FUNCTION_BLOCK INTERNAL FB_State3 EXTENDS FB_State
VAR_INPUT
END_VAR
VAR_OUTPUT
END_VAR
VAR
END_VAR

END_FUNCTION_BLOCK

(* stored: Version 1.1.0.1, ProductVersion 3.1.4024.12
   POU FB_State3: Id {746f3b1a-34f3-0ad3-0d50-0dde032c9dbf}, SpecialFunc None *)
